// TIA Portal V16 export
// export: Created 2021-06-25T07:11:59.4299352Z, ExportSetting WithDefaults, DisplayName Totally Integrated Automation Portal, DisplayVersion V16, DisplayName TIA Portal Version Control Interface, DisplayVersion V16, DisplayName TIA Portal Openness, DisplayVersion V16, DisplayName STEP 7 Professional, DisplayVersion V16, DisplayName STEP 7 Safety, DisplayVersion V16, DisplayName WinCC Advanced, DisplayVersion V16
ORGANIZATION_BLOCK "Main"   // OB1, LAD, ProgramCycle
TITLE = "Main Program Sweep (Cycle)"
{ S7_Optimized_Access := 'TRUE' }
VERSION : 0.1
// stored: AutoNumber true, IsIECCheckEnabled false, SetENOAutomatically false
   VAR_INPUT
      Initial_Call : Bool;   // Initial call of this OB
      Remanence : Bool;   // =True, if remanent data are available
   END_VAR
   VAR_TEMP
      RES : Bool;
   END_VAR
BEGIN

REGION Network 1
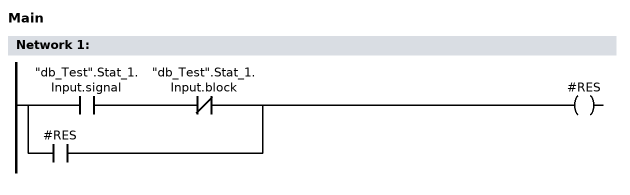
   RUNG wire#powerrail
      Contact( "db_Test".Stat_1.Input.signal )
      I_Contact( "db_Test".Stat_1.Input.block )
      wire#w1
      Coil( #RES )
   END_RUNG
   RUNG wire#powerrail
      Contact( #RES )
   END_RUNG wire#w1
   // the same network as SCL:
   #RES := ("db_Test".Stat_1.Input.signal AND NOT "db_Test".Stat_1.Input.block) OR #RES;
END_REGION
END_ORGANIZATION_BLOCK
